TYPE ST_RemovePathData :
STRUCT
	sObjectID					: STRING := 'MAIN.fbMMServer';
	sMethodID					: STRING := 'MAIN.fbMMServer#M_RemovePath';
	iStatus						: INT;
	iNoOfInputArgs				: BYTE := 2;
	iNoOfOutputArgs				: BYTE := 2;
	stInput						: ST_RemovePathDataIn;
	stOutput					: ST_RemovePathDataOut;	
END_STRUCT
END_TYPE

(* stored: Version 1.1.0.1, ProductVersion 3.1.4024.5
   DUT ST_RemovePathData: Id {54357481-2be7-481e-98f2-118ba0e16f7b} *)
